(* PLC project KinIn_v3.project, CODESYS CODESYS V3.5 SP19 *)
(* stored: creationDateTime 2025-01-20T16:23:18.8896075, modificationDateTime 2025-01-20T16:17:39.6822999 *)

FUNCTION_BLOCK BodyJacobian
  VAR_INPUT
    {attribute 'variable_length_array_original_scope' := 'Inout'}
    {attribute 'variable_length_array' := 'ARRAY[*,*] OF REAL'}
    {attribute 'Dimensions' := '2'}
    Blist : POINTER TO REAL;
    {attribute 'variable_length_array_original_scope' := 'Inout'}
    {attribute 'variable_length_array' := 'ARRAY[*] OF REAL'}
    {attribute 'Dimensions' := '1'}
    thetalist : POINTER TO REAL;
    {attribute 'variable_length_array_original_scope' := 'Inout'}
    {attribute 'variable_length_array' := 'ARRAY[*,*] OF REAL'}
    {attribute 'Dimensions' := '2'}
    Jb : POINTER TO REAL;  (* 6xnt nt: number of theta *)
  END_VAR
  VAR
    MatMul : MatMul;
    Eye : Eye;
    spatialVelToSE3Matrix : spatialVelToSE3Matrix;
    TransSE3_fromExp_se3 : TransSE3_fromExp_se3;
    AdjointTransform : AdjointTransform;
    i : DINT;
    j : DINT;
    T : ARRAY[1..4, 1..4] OF REAL;
    T_inside : ARRAY[1..6] OF REAL;  (* temporal variables *)
    se3mat : ARRAY[1..4, 1..4] OF REAL;
    T_exp6 : ARRAY[1..4, 1..4] OF REAL;
    T_product : ARRAY[1..4, 1..4] OF REAL;
    AdT : ARRAY[1..6, 1..6] OF REAL;
    i1 : DINT;
    j1 : DINT;
    Jb_temp : ARRAY[1..6, 1..6] OF REAL;
  END_VAR

            i:=1;j:=1;
FOR i:=1 TO UPPER_BOUND(Blist,1) DO
	FOR j:=1 TO UPPER_BOUND(Blist,2) DO
		Jb[i,j]:=Blist[i,j];
	END_FOR
END_FOR

Eye(eye:= T);

i:=UPPER_BOUND(thetalist,1)-1;
FOR i:=UPPER_BOUND(thetalist,1)- 1 TO 1 BY -1 DO
	//T_inside:=-1 * Blist(:, i + 1) * thetalist(i + 1)
	j:=1;
	FOR j:=1 TO UPPER_BOUND(Blist,1) DO
		T_inside[j]:=-1 * Blist[j, i + 1] * thetalist[i + 1];
	END_FOR
	//T = T * MatrixExp6(VecTose3(T_inside));
	spatialVelToSE3Matrix(V:=T_inside , se3mat=> se3mat);
	TransSE3_fromExp_se3(se3mat:=se3mat , T=> T_exp6);
	MatMul(mat1:=T , mat2:=T_exp6 , MatResult:= T_product);
	
	i1:=1;j1:=1;//assign again T for the next iteration
	FOR i1:=1 TO 4 DO//until 4
		FOR j1:=1 TO 4 DO//until 4
			T[i1,j1]:=T_product[i1,j1];
		END_FOR
	END_FOR
	//Jb(:, i) = Adjoint(T) * Blist(:, i);
	AdjointTransform(Transform4x4:= T_product, AdT=>AdT );
	
	//Jb[k,i]:=0;	Already initialized similar to Blist
	i1:=1;j1:=1;
	FOR i1:=1 TO UPPER_BOUND(Jb,1) DO//until 6
		Jb[i1,i]:=0;//the not affected equal Blist
		Jb_temp[i1,i]:=0;
		FOR j1:=1 TO UPPER_BOUND(Jb,1) DO //always 6 too
			Jb[i1,i]:=Jb[i1,i]+AdT[i1,j1]*Blist[j1,i];
			Jb_temp[i1,i]:=Jb[i1,i]+AdT[i1,j1]*Blist[j1,i];
		END_FOR
	END_FOR
END_FOR
          
END_FUNCTION_BLOCK
